{attribute 'qualified_only'}
{attribute 'strict'}
TYPE E_ProgramState :
(
	INIT,
	REFRESH_SETPOINTS_USING_FORMULA,
	WAIT_FOR_START_COMMAND,
	ACTIVE,
	COMPLETE,
	RESET	
);
END_TYPE

(* stored: Version 1.1.0.1, ProductVersion 3.1.4024.0
   DUT E_ProgramState: Id {75ce36ce-63fb-42dc-8544-0e422db8040f} *)
